FUNCTION_BLOCK FB_CSVEventStorage IMPLEMENTS EventStorage
VAR 
	// Enum for state machine
	eWriteState: (	FILE_OPEN_TRIGGER,FILE_OPEN,WAIT_FOR_EVENT,WRITE_EVENT_TRIGGER,
					WRITE_EVENT,FILE_CLOSE_TRIGGER, FILE_CLOSE,ERROR);
				 
	fbFileOpen: FB_FileOpen := (bExecute := FALSE, sPathName := 'C:\Events.log', nMode := FOPEN_MODEAPPEND OR FOPEN_MODETEXT);
	
	fbFilePuts: FB_FilePuts();
	fbFileClose: FB_FileClose();

	stWriteEvent: ST_EVENT; // The st_event which is supposed to be written	
	csvString: T_MaxString;
END_VAR

CASE eWriteState OF
	
	FILE_OPEN_TRIGGER :
		// Start the function, the rising edge is started and the function will be continously called 
		// until windows allows it to be opened
		fbFileOpen(bExecute:= TRUE);
		eWriteState := FILE_OPEN;
		
	FILE_OPEN :
		fbFileOpen(bExecute:= FALSE);
		IF fbFileOpen.bError THEN
			eWriteState := ERROR; // You can also do something like rerunning the above to check again
		ELSIF NOT fbFileOpen.bBusy AND fbFileOpen.hFile <> 0 THEN
			 eWriteState := WAIT_FOR_EVENT;
		END_IF
	
	WAIT_FOR_EVENT :
		// Do Nothing here see StoreEvent
	
	WRITE_EVENT_TRIGGER:
		csvString := STEventToCSVString(stEvent := stWriteEvent);
		fbFilePuts(bExecute:= FALSE);
		fbFilePuts(bExecute:= TRUE, sLine := csvString, hFile := fbFileOpen.hFile);
		eWriteState := WRITE_EVENT;
	
	WRITE_EVENT :
		fbFilePuts(bExecute:= FALSE);
		IF fbFilePuts.bError THEN
			eWriteState := Error;
		ELSIF NOT fbFilePuts.bBusy THEN
			// This was for when we had to coninously wait for new writes in storeEVent method
			// But it wouldn't write as the file had to be closed
			// eWriteState:= WAIT_FOR_EVENT; 
			
			eWriteState:= FILE_CLOSE_TRIGGER;
		END_IF
		
	
	FILE_CLOSE_TRIGGER: 
		fbFileClose(bExecute := FALSE);
		fbFileClose(bExecute := TRUE, hFile :=fbFileOpen.hFile);
		eWriteState := FILE_CLOSE;
		
	FILE_CLOSE :
		fbFileClose(bExecute := FALSE);
		IF fbFileClose.bError THEN
			eWriteState := Error;
		ELSIF NOT fbFileClose.bBusy THEN
			eWriteState := FILE_OPEN_TRIGGER;
		END_IF
	
	ERROR :
		fbFileOpen.nErrId;
	
END_CASE

METHOD PRIVATE STEventToCSVString: T_MaxString
VAR_INPUT
	stEvent : REFERENCE TO ST_EVENT;
END_VAR
VAR
	stringHolder: T_MaxString;
END_VAR
stringHolder := TO_STRING(stEvent.eEventType); // This works because of the attribute added to the enum
stringHolder := CONCAT(str1 := stringHolder, str2 := ',');

stringHolder := CONCAT(str1 := stringHolder, str2 := TO_STRING(stEvent.eEventSeverity)); // Here only numbers will be added
stringHolder := CONCAT(str1 := stringHolder, str2 := ',');

stringHolder := CONCAT(str1 := stringHolder, str2 := TO_STRING(stEvent.nEventId));
stringHolder := CONCAT(str1 := stringHolder, str2 := ',');

stringHolder := CONCAT(str1 := stringHolder, str2 := F_RTRIM(stEvent.sEventText));
stringHolder := CONCAT(str1 := stringHolder, str2 := ',');

stringHolder := CONCAT(str1 := stringHolder, str2 := TO_STRING(stEvent.dtTimeStamp));
stringHolder := CONCAT(str1 := stringHolder, str2 := '$n'); // New line

STEventToCSVString := stringHolder;
END_METHOD

// add method implementation 
METHOD StoreEvent
VAR_INPUT
	st_event	: ST_Event;
END_VAR
IF eWriteState = WAIT_FOR_EVENT THEN
	eWriteState := WRITE_EVENT_TRIGGER;
	stWriteEvent:= st_event;
END_IF
END_METHOD

END_FUNCTION_BLOCK

(* stored: Version 1.1.0.1, ProductVersion 3.1.4024.12
   POU FB_CSVEventStorage: Id {f353186e-7405-4515-8068-9da4b6365fa3}, SpecialFunc None
   Method STEventToCSVString: Id {8b6c81ef-06b6-4710-a9f7-053a54dfe41d}
   Method StoreEvent: Id {2010f449-e83a-464f-a1c0-9ccf79d9cd0a} *)
